{attribute 'qualified_only'}
VAR_GLOBAL
//Output from process to PLC
	qxStrobe		AT %Q*:	BOOL;
	qxDir			AT %Q*:	INT;
	
//Input to process from PLC
	iiAtStation1		AT %I*:	BOOL;
	iiAtStation2		AT %I*:	BOOL;
END_VAR

(* stored: Version 1.1.0.1, ProductVersion 3.1.4024.12
   GVL GVL: Id {71d90b3b-838f-42b7-9031-672ba951413e} *)
